FUNCTION_BLOCK NodeFactoryCollection IMPLEMENTS I_NodeFactoryCollection
VAR
	nodeFactories : Dictionary;
END_VAR

METHOD PUBLIC GetByType : I_NodeFactory
VAR_INPUT
	NodeType : T_MAXSTRING;
END_VAR
nodeFactories.TryGetValue(NodeType, GetByType);
END_METHOD

METHOD PUBLIC HasType : BOOL
VAR_INPUT
	NodeType : T_MAXSTRING;
END_VAR
nodeFactories.ContainsKey(NodeType);
END_METHOD

METHOD PUBLIC InsertByType
VAR_INPUT
	NodeType : T_MAXSTRING;
	NodeFactory : I_NodeFactory;
END_VAR
nodeFactories.AddOrUpdate(NodeType, NodeFactory);
END_METHOD

END_FUNCTION_BLOCK

(* stored: Version 1.1.0.1, ProductVersion 3.1.4024.12
   POU NodeFactoryCollection: Id {3a71411c-013f-04b4-2fdb-abd75ba10395}, SpecialFunc None
   Method GetByType: Id {ca3ebbc1-de44-0bf3-2840-81a4910c38fe}
   Method HasType: Id {2598df50-d563-0c6e-0aca-47ba8cbbf0c4}
   Method InsertByType: Id {4d3a5f0c-8074-09fb-2906-a4aa05ab5434} *)
